PROGRAM Laser
VAR
END_VAR

END_PROGRAM

(* stored: Version 1.1.0.1, ProductVersion 3.1.4024.12
   POU Laser: Id {5724ed8c-95a4-443b-8d0a-229c2f523827}, SpecialFunc None *)
